# EPICS substitutions: ek9000App/Db/EL3144.substitutions
file EL3144.template
{       pattern
        {
                TERMINAL,

        }
        {
        }
}
